INTERFACE I_ULINT EXTENDS I_Datatype

PROPERTY PUBLIC Value : REFERENCE TO ULINT
GET
END_GET
END_PROPERTY

END_INTERFACE

(* stored: Version 1.1.0.1, ProductVersion 3.1.4024.15
   Itf I_ULINT: Id {3ebc358f-1f13-0940-2bd8-78a9aa1abb01}
   Property Value: Id {82e3b063-9aea-0c67-2273-1eaefdd4db3a}
   Get Get: Id {78fe9476-ab02-0f6a-01e5-d0a60f94ce07} *)
